// TIA Portal V20 export
DATA_BLOCK "InstMemCardDiag"   // DB122
AUTHOR : Siemens Digital Industries
FAMILY : LAF
// stored: AssignedProDiagFB ProDiag, InstanceOfName LAF_MemCardDiag, InstanceOfType FB
"LAF_MemCardDiag"
   // VAR_INPUT
   //    plantIdentifier { ExternalAccessible := 'False'; ExternalVisible := 'False'; ExternalWritable := 'False'} : WString[24] := WSTRING#'SMC_Diagnostic';
   //    textListId { ExternalAccessible := 'False'; ExternalVisible := 'False'; ExternalWritable := 'False'} : Int := 585;
   //    firstCycle { ExternalAccessible := 'False'; ExternalVisible := 'False'; ExternalWritable := 'False'} : Bool := FALSE;
   //    readInfoMemCard { ExternalAccessible := 'False'; ExternalVisible := 'False'; ExternalWritable := 'False'} : Bool := FALSE;
   //    hideAlarmMask { ExternalAccessible := 'False'; ExternalVisible := 'False'; ExternalWritable := 'False'} : Byte := 16#00;
   // END_VAR
   // VAR_OUTPUT
   //    generalAlarm { ExternalAccessible := 'False'; ExternalVisible := 'False'; ExternalWritable := 'False'} : Bool := FALSE;
   //    generalWarn { ExternalAccessible := 'False'; ExternalVisible := 'False'; ExternalWritable := 'False'} : Bool := FALSE;
   //    generalInfo { ExternalAccessible := 'False'; ExternalVisible := 'False'; ExternalWritable := 'False'} : Bool := FALSE;
   // END_VAR
   // VAR_IN_OUT
   //    diagHmi : "LAF_typeMemCardDiag";
   // END_VAR
   // VAR
   //    statMessages { ExternalAccessible := 'False'; ExternalVisible := 'False'; ExternalWritable := 'False'} : "LAF_typeMemCardMessages";
   //    statHideMessages { ExternalAccessible := 'False'; ExternalVisible := 'False'; ExternalWritable := 'False'} : "LAF_typeMemCardMessages";
   //    statStep { ExternalAccessible := 'False'; ExternalVisible := 'False'; ExternalWritable := 'False'} : Array[0..3] of Bool;
   //    statRisEdgeStep0 { ExternalAccessible := 'False'; ExternalVisible := 'False'; ExternalWritable := 'False'} : Bool := FALSE;
   //    statRisEdgeStep1 { ExternalAccessible := 'False'; ExternalVisible := 'False'; ExternalWritable := 'False'} : Bool := FALSE;
   //    statAlarmNo { ExternalAccessible := 'False'; ExternalVisible := 'False'; ExternalWritable := 'False'} : UInt := 99;
   //    statWarnNo { ExternalAccessible := 'False'; ExternalVisible := 'False'; ExternalWritable := 'False'} : UInt := 99;
   //    statInfoNo { ExternalAccessible := 'False'; ExternalVisible := 'False'; ExternalWritable := 'False'} : UInt := 99;
   //    instGetInfoMode0 { ExternalAccessible := 'False'; ExternalVisible := 'False'; ExternalWritable := 'False'} : GetSMCinfo;
   //    instGetInfoMode1 { ExternalAccessible := 'False'; ExternalVisible := 'False'; ExternalWritable := 'False'} : GetSMCinfo;
   //    instGetInfoMode2 { ExternalAccessible := 'False'; ExternalVisible := 'False'; ExternalWritable := 'False'} : GetSMCinfo;
   //    instGetInfoMode3 { ExternalAccessible := 'False'; ExternalVisible := 'False'; ExternalWritable := 'False'} : GetSMCinfo;
   // END_VAR
BEGIN
   statMessages.invalidValueModeParam := FALSE;
   statMessages.noMemCardInserted := FALSE;
   statMessages.noDataAvailable := FALSE;
   statMessages.maxCallsReached := FALSE;
   statMessages.configMemSpaceWarning := FALSE;
   statMessages.configMemSpaceAlarm := FALSE;
   statMessages.usedLiftetimeInvalid := FALSE;
   statMessages.diagAlarmDisabled := FALSE;
   statHideMessages.invalidValueModeParam := FALSE;
   statHideMessages.noMemCardInserted := FALSE;
   statHideMessages.noDataAvailable := FALSE;
   statHideMessages.maxCallsReached := FALSE;
   statHideMessages.configMemSpaceWarning := FALSE;
   statHideMessages.configMemSpaceAlarm := FALSE;
   statHideMessages.usedLiftetimeInvalid := FALSE;
   statHideMessages.diagAlarmDisabled := FALSE;
   statStep[0..3] := FALSE;
   instGetInfoMode0.REQ := FALSE;
   instGetInfoMode0.Mode := 0;
   instGetInfoMode0.Done := FALSE;
   instGetInfoMode0.Busy := FALSE;
   instGetInfoMode0.Error := FALSE;
   instGetInfoMode0.Status := 16#7000;
   instGetInfoMode0.Info := 31151664;
   instGetInfoMode1.REQ := FALSE;
   instGetInfoMode1.Mode := 1;
   instGetInfoMode1.Done := FALSE;
   instGetInfoMode1.Busy := FALSE;
   instGetInfoMode1.Error := FALSE;
   instGetInfoMode1.Status := 16#7000;
   instGetInfoMode1.Info := 68208;
   instGetInfoMode2.REQ := FALSE;
   instGetInfoMode2.Mode := 2;
   instGetInfoMode2.Done := FALSE;
   instGetInfoMode2.Busy := FALSE;
   instGetInfoMode2.Error := FALSE;
   instGetInfoMode2.Status := 16#7000;
   instGetInfoMode2.Info := 0;
   instGetInfoMode3.REQ := FALSE;
   instGetInfoMode3.Mode := 3;
   instGetInfoMode3.Done := FALSE;
   instGetInfoMode3.Busy := FALSE;
   instGetInfoMode3.Error := FALSE;
   instGetInfoMode3.Status := 16#7000;
   instGetInfoMode3.Info := 80;
END_DATA_BLOCK
